// TwinCAT 3 PLC project Monolitico
// ProgramVersion: 3.1.4024.0
// libraries:
//   CmpBitmapPool, * (System)
//   Tc2_Standard, * (Beckhoff Automation GmbH)
//   Tc2_System, * (Beckhoff Automation GmbH)
//   Tc3_Module, * (Beckhoff Automation GmbH)
//   VisuDialogs, * (System)
// project tree:
//   / GlobalTextList.TcGTLO, PlcTask.TcTTO, Visualization Manager.TcVMO (not stored)
//   POUs/ FB_Bloque.TcPOU, MAIN.TcPOU
//   VISUs/ ImagePool.TcIPO (not stored), Visualization.TcVIS
// (motion and I/O tree: see PLC project manual)
// real-time tasks:
//   TASK PlcTask: cycle T#10ms, priority 20, ADS port 350
//   TASK PlcTask1: cycle T#10ms, priority 21, ADS port 351

CONFIGURATION Monolitico
    RESOURCE PLC ON TwinCAT3
        TASK PlcTask(INTERVAL := T#10ms, PRIORITY := 20);
        PROGRAM MAIN WITH PlcTask : MAIN;
    END_RESOURCE
END_CONFIGURATION

// ---- POUs/MAIN.TcPOU
PROGRAM MAIN
VAR
	
	//Pulsador AT %I*: BOOL;
	//Lampara AT %Q*: BOOL;
	
	Selector_modo_manual AT %I*: BOOL;
	
	test_pieza: FB_Bloque;

END_VAR

IF NOT Selector_modo_manual THEN
test_pieza();
END_IF

END_PROGRAM

// ---- POUs/FB_Bloque.TcPOU
FUNCTION_BLOCK FB_Bloque
VAR_INPUT
	Tcheck: TIME := T#1S;
	Treset: TIME := T#1S;
	Tdesplazador: TIME := T#1S;
	Tcinta: TIME := T#0.5S;
END_VAR
VAR_OUTPUT
END_VAR
VAR
	Ciclos: INT;
	Aceptados:INT;
	Rechazados: INT;
	Restantes: INT;
	
	pieza_ok: BOOL;
	
	//Terminal 2
	Pulsador_parada_emergencia AT %I*: BOOL;
	Selector_modo_manual AT %I*: BOOL;
	Pulsador_marcha AT %I*: BOOL;
	Pulsador_parada_NC AT %I*: BOOL;
	Parte_operativa_conectada AT %I*: BOOL;
	Presencia_pale AT %I*: BOOL;
	Codigo_pale_bit_0 AT %I*: BOOL;
	Codigo_pale_bit_1 AT %I*: BOOL;
	
	
	//Terminal 3
	Codigo_pale_bit_2 AT %I*: BOOL;
	Detector_presion AT %I*: BOOL;
	
	//Terminal 4
	Desconecta_parte_operativa AT %Q*: BOOL;
	Lampara_alarma AT %Q*: BOOL;
	Lampara_marcha AT %Q*: BOOL;
	Lampara_falta_material AT %Q*: BOOL;
	Activa_marcha_motor_cinta AT %Q*: BOOL;
	Invierte_marcha_motor_cinta AT %Q*: BOOL;
	Retenedor_pale_baja AT %Q*: BOOL;
	Separador_pale_sube AT %Q*: BOOL;
	
	
	//Terminal 5
 	Avisador_sonoro AT %Q*: BOOL;
	
	//Terminal 6
	Horizontal_descargador_detras AT %I*: BOOL;
	Horizontal_descargador_delante AT %I*: BOOL;
	Vertical_descargador_arriba AT %I*: BOOL;
	Vertical_descargador_abajo AT %I*: BOOL;
	Verificador_arriba AT %I*: BOOL;
	Verificador_abajo AT %I*: BOOL;
	Desplazador_detras AT %I*: BOOL;
	Alimentador_detras AT %I*: BOOL;
	
	
	//Terminal 7
	Alimentador_delante AT %I*: BOOL;
	Vacio_obtenido_vacuostato_descargador AT %I*: BOOL;
	Base_en_Alimentador AT %I*: BOOL;
	
	//Terminal 8
	Descargador_adelante AT %Q*: BOOL;
	Descargador_atras AT %Q*: BOOL;
	Descargador_baja AT %Q*: BOOL;
	Rechazador_adelante AT %Q*: BOOL;
	Verificador_baja AT %Q*: BOOL;
	Desplazador_adelante AT %Q*: BOOL;
	Alimentador_adelante AT %Q*: BOOL;
	Eyector_succiona AT %Q*: BOOL;
	
	NOLAMP: INT;
	t: INT;
	NOTSOUND: INT;
	NOTFOUND: INT;
END_VAR

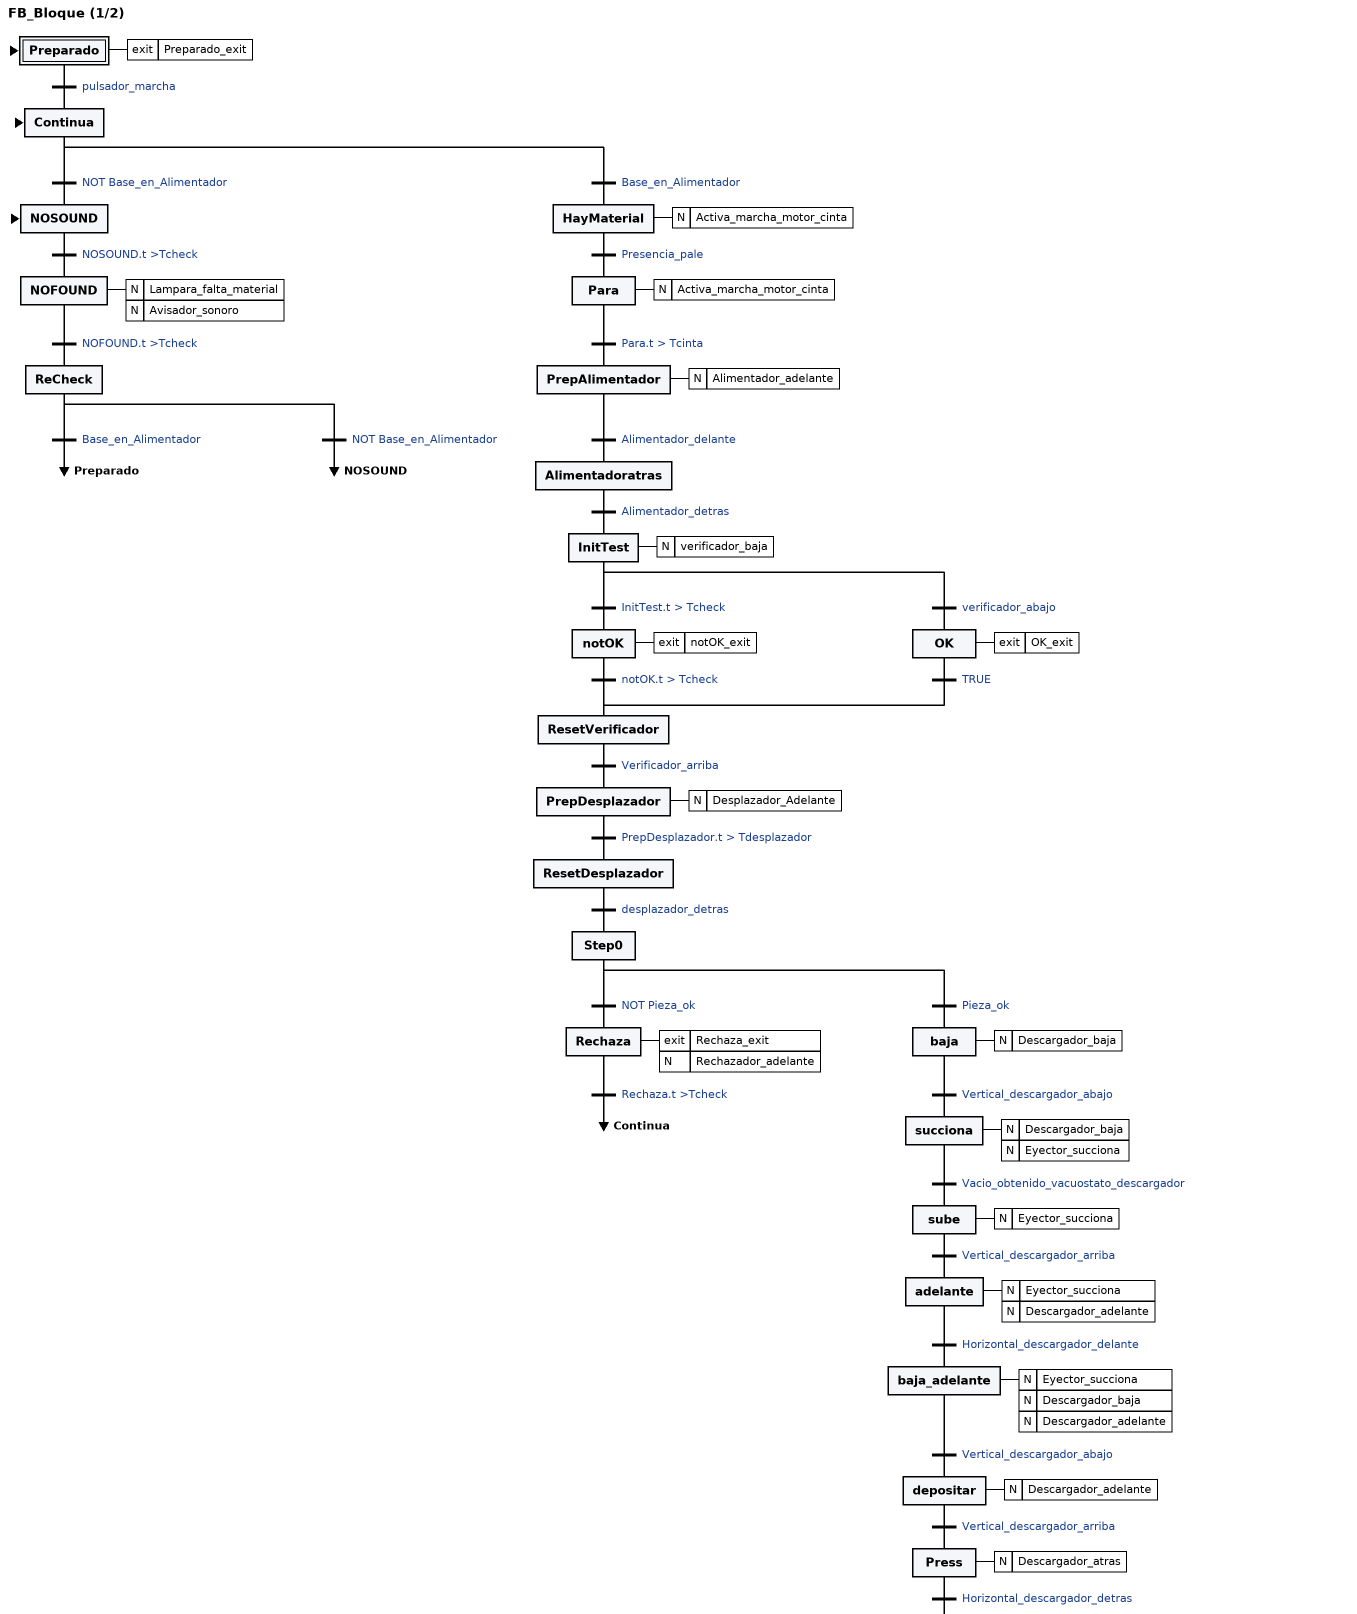
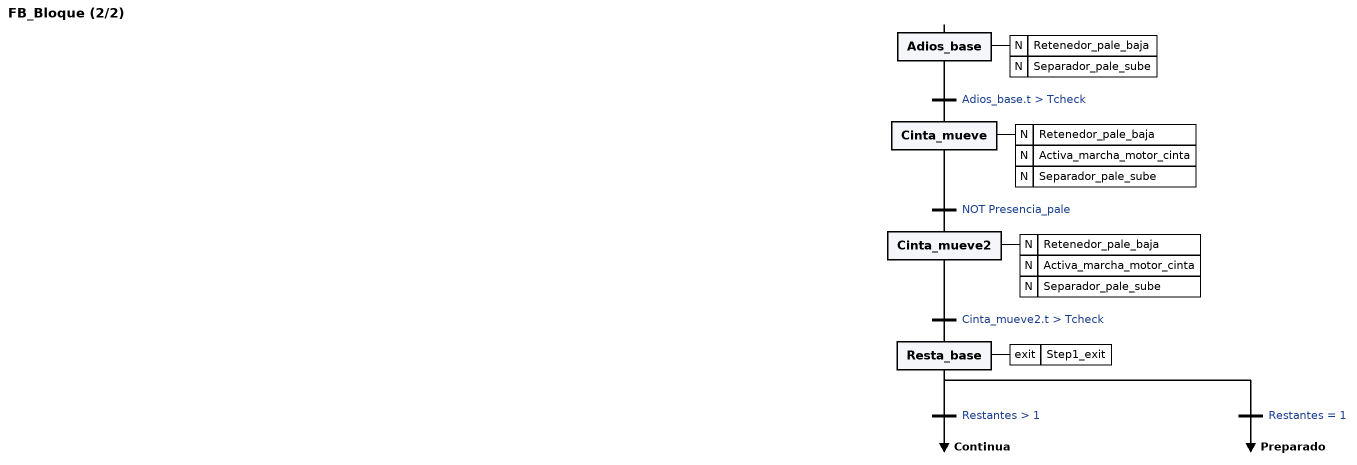
INITIAL_STEP Preparado:
    Preparado_exit(P0);  // exit action
END_STEP
TRANSITION FROM Preparado TO Continua
    := pulsador_marcha;
END_TRANSITION
STEP Continua:
END_STEP
TRANSITION FROM Continua TO NOSOUND
    := NOT Base_en_Alimentador;
END_TRANSITION
STEP NOSOUND:
END_STEP
TRANSITION FROM NOSOUND TO NOFOUND
    := NOSOUND.t >Tcheck;
END_TRANSITION
STEP NOFOUND:
    Lampara_falta_material(N);
    Avisador_sonoro(N);
END_STEP
TRANSITION FROM NOFOUND TO ReCheck
    := NOFOUND.t >Tcheck;
END_TRANSITION
STEP ReCheck:
END_STEP
TRANSITION FROM ReCheck TO Preparado
    := Base_en_Alimentador;
END_TRANSITION
TRANSITION FROM ReCheck TO NOSOUND
    := NOT Base_en_Alimentador;
END_TRANSITION
TRANSITION FROM Continua TO HayMaterial
    := Base_en_Alimentador;
END_TRANSITION
STEP HayMaterial:
    Activa_marcha_motor_cinta(N);
END_STEP
TRANSITION FROM HayMaterial TO Para
    := Presencia_pale;
END_TRANSITION
STEP Para:
    Activa_marcha_motor_cinta(N);
END_STEP
TRANSITION FROM Para TO PrepAlimentador
    := Para.t > Tcinta;
END_TRANSITION
STEP PrepAlimentador:
    Alimentador_adelante(N);
END_STEP
TRANSITION FROM PrepAlimentador TO Alimentadoratras
    := Alimentador_delante;
END_TRANSITION
STEP Alimentadoratras:
END_STEP
TRANSITION FROM Alimentadoratras TO InitTest
    := Alimentador_detras;
END_TRANSITION
STEP InitTest:
    verificador_baja(N);
END_STEP
TRANSITION FROM InitTest TO notOK
    := InitTest.t > Tcheck;
END_TRANSITION
STEP notOK:
    notOK_exit(P0);  // exit action
END_STEP
TRANSITION FROM notOK TO ResetVerificador
    := notOK.t > Tcheck;
END_TRANSITION
TRANSITION FROM InitTest TO OK
    := verificador_abajo;
END_TRANSITION
STEP OK:
    OK_exit(P0);  // exit action
END_STEP
TRANSITION FROM OK TO ResetVerificador
    := TRUE;
END_TRANSITION
STEP ResetVerificador:
END_STEP
TRANSITION FROM ResetVerificador TO PrepDesplazador
    := Verificador_arriba;
END_TRANSITION
STEP PrepDesplazador:
    Desplazador_Adelante(N);
END_STEP
TRANSITION FROM PrepDesplazador TO ResetDesplazador
    := PrepDesplazador.t > Tdesplazador;
END_TRANSITION
STEP ResetDesplazador:
END_STEP
TRANSITION FROM ResetDesplazador TO Step0
    := desplazador_detras;
END_TRANSITION
STEP Step0:
END_STEP
TRANSITION FROM Step0 TO Rechaza
    := NOT Pieza_ok;
END_TRANSITION
STEP Rechaza:
    Rechaza_exit(P0);  // exit action
    Rechazador_adelante(N);
END_STEP
TRANSITION FROM Rechaza TO Continua
    := Rechaza.t >Tcheck;
END_TRANSITION
TRANSITION FROM Step0 TO baja
    := Pieza_ok;
END_TRANSITION
STEP baja:
    Descargador_baja(N);
END_STEP
TRANSITION FROM baja TO succiona
    := Vertical_descargador_abajo;
END_TRANSITION
STEP succiona:
    Descargador_baja(N);
    Eyector_succiona(N);
END_STEP
TRANSITION FROM succiona TO sube
    := Vacio_obtenido_vacuostato_descargador;
END_TRANSITION
STEP sube:
    Eyector_succiona(N);
END_STEP
TRANSITION FROM sube TO adelante
    := Vertical_descargador_arriba;
END_TRANSITION
STEP adelante:
    Eyector_succiona(N);
    Descargador_adelante(N);
END_STEP
TRANSITION FROM adelante TO baja_adelante
    := Horizontal_descargador_delante;
END_TRANSITION
STEP baja_adelante:
    Eyector_succiona(N);
    Descargador_baja(N);
    Descargador_adelante(N);
END_STEP
TRANSITION FROM baja_adelante TO depositar
    := Vertical_descargador_abajo;
END_TRANSITION
STEP depositar:
    Descargador_adelante(N);
END_STEP
TRANSITION FROM depositar TO Press
    := Vertical_descargador_arriba;
END_TRANSITION
STEP Press:
    Descargador_atras(N);
END_STEP
TRANSITION FROM Press TO Adios_base
    := Horizontal_descargador_detras;
END_TRANSITION
STEP Adios_base:
    Retenedor_pale_baja(N);
    Separador_pale_sube(N);
END_STEP
TRANSITION FROM Adios_base TO Cinta_mueve
    := Adios_base.t > Tcheck;
END_TRANSITION
STEP Cinta_mueve:
    Retenedor_pale_baja(N);
    Activa_marcha_motor_cinta(N);
    Separador_pale_sube(N);
END_STEP
TRANSITION FROM Cinta_mueve TO Cinta_mueve2
    := NOT Presencia_pale;
END_TRANSITION
STEP Cinta_mueve2:
    Retenedor_pale_baja(N);
    Activa_marcha_motor_cinta(N);
    Separador_pale_sube(N);
END_STEP
TRANSITION FROM Cinta_mueve2 TO Resta_base
    := Cinta_mueve2.t > Tcheck;
END_TRANSITION
STEP Resta_base:
    Step1_exit(P0);  // exit action
END_STEP
TRANSITION FROM Resta_base TO Continua
    := Restantes > 1;
END_TRANSITION
TRANSITION FROM Resta_base TO Preparado
    := Restantes = 1;
END_TRANSITION

ACTION notOK_exit:
pieza_ok := FALSE;
END_ACTION

ACTION OK_exit:
pieza_ok := true;
END_ACTION

ACTION Preparado_entry:
//Ciclos:= 3;
Rechazados :=0;
Aceptados :=0;
Restantes:=Ciclos;
END_ACTION

ACTION Preparado_exit:
IF Restantes = 0 THEN

	Restantes := Ciclos;
	Aceptados := 0;
	Rechazados := 0;	

END_IF
END_ACTION

ACTION Rechaza_exit:
Rechazados:= Rechazados+1;
END_ACTION

ACTION Step1_exit:
Aceptados:=Aceptados+1;
Restantes:=Restantes-1;
END_ACTION

END_FUNCTION_BLOCK

// ---- GlobalTextList.TcGTLO
TEXTLIST GlobalTextList
  189 = '  ➡ ⬅ ⬇ ⬆ ← → ↓ ↑'
  198 = ' ➙'
  307 = '%i'
  729 = '0'
  472 = '1'
  731 = '<'
  44 = '>'
  12 = 'A+'
  482 = 'A-'
  789 = 'Abajo'
  231 = 'Aceptados'
  66 = 'Alarma'
  224 = 'Alimentador'
  25 = 'Arriba'
  54 = 'Aspirar'
  267 = 'B+'
  782 = 'B-'
  801 = 'C+'
  215 = 'C-'
  701 = 'Ciclos'
  642 = 'Ciclos Completados'
  957 = 'Cinta'
  81 = 'Colocado'
  497 = 'Comenzar'
  143 = 'D+'
  630 = 'D-'
  481 = 'Delante'
  437 = 'Descargador'
  936 = 'Desplazador'
  445 = 'Detrás'
  74 = 'E+'
  781 = 'E-'
  742 = 'E-Stop'
  908 = 'Estado'
  286 = 'Estoy Abajo'
  148 = 'Estoy Arriba'
  955 = 'Eyector'
  417 = 'F+'
  707 = 'F-'
  878 = 'FALTA M.'
  395 = 'FM'
  769 = 'FMS-201                                 ALIMENTADORA DE BASES                                                    VTL     '
  561 = 'Horizontal'
  750 = 'Lámpara'
  45 = 'Marcha'
  634 = 'Material'
  861 = 'Panel'
  463 = 'Parada'
  619 = 'pb'
  935 = 'Pieza NO OK'
  336 = 'Pieza OK'
  741 = 'Pieza Ok'
  524 = 'Planta'
  640 = 'pp'
  783 = 'Preparado'
  330 = 'R+'
  876 = 'Rechazador'
  970 = 'Rechazados'
  888 = 'Rechazads'
  94 = 'Rehczados'
  560 = 'Restantes'
  531 = 'Rev'
  452 = 'Run'
  784 = 'S+'
  815 = 'Succionar'
  643 = 'Tarea'
  710 = 'V+'
  288 = 'V-'
  629 = 'Vacío'
  125 = 'Verificador'
  839 = 'Verificador Activado'
  483 = 'Vertical'
  575 = '➡'
  509 = '⬅'
  381 = '⬆'
  169 = '⬇'
END_TEXTLIST

// ---- VISUs/Visualization.TcVIS
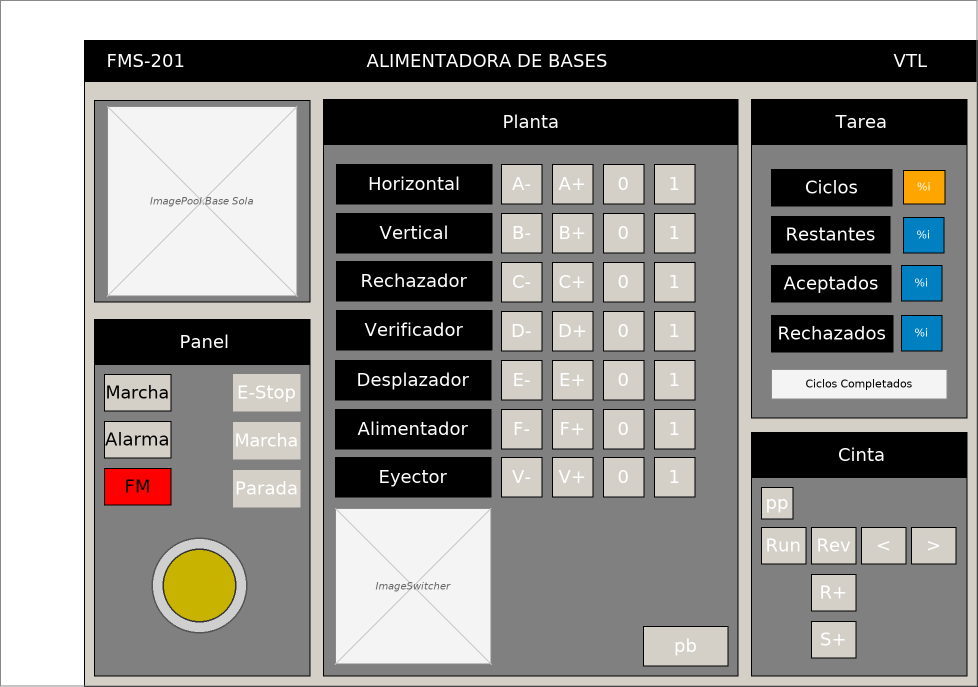
VISUALIZATION Visualization  // 978x687
    Rectangle (84,81 894x606)
    Rectangle (751,144 216x274)
    Rectangle (323,144 415x532)
    Rectangle (323,99 415x45)
    Label (323,101 416x42), "Planta"
    Rectangle (751,99 216x45)
    Label (801,104 121x36), "Tarea"
    Progressbar (771,369 176x30), "Ciclos Completados", variable: MAIN.test_pieza.Aceptados
    RoundedRectangle (336,164 156x40), "Horizontal", colour toggle: MAIN.test_pieza.Descargador_adelante
    Textfield (903,170 42x34), "%i", text variable: MAIN.test_pieza.Ciclos
        OnMouseDown: write MAIN.test_pieza.Ciclos via VisuDialogs.Numpad, min 1, max 10
    RoundedRectangle (771,169 121x37), "Ciclos"
    RoundedRectangle (771,216 119x37), "Restantes"
    RoundedRectangle (771,265 120x37), "Aceptados"
    RoundedRectangle (771,315 122x37), "Rechazados"
    Textfield (903,217 41x36), "%i", text variable: MAIN.test_pieza.Restantes
    Textfield (901,265 41x36), "%i", text variable: MAIN.test_pieza.Aceptados
    Textfield (901,315 41x36), "%i", text variable: MAIN.test_pieza.Rechazados
    RoundedRectangle (552,213 41x40), "B+", colour toggle: MAIN.test_pieza.Descargador_baja
        toggle MAIN.test_pieza.Descargador_baja
    Rectangle (751,477 216x199)
    Rectangle (751,432 216x45)
    Label (801,437 121x36), "Cinta"
    Rectangle (94,100 216x202)
    Rectangle (94,364 216x312)
    Rectangle (94,319 216x45)
    Label (144,324 121x36), "Panel"
    Rectangle (84,40 894x41)
    Label (84,41 893x40), "FMS-201 ALIMENTADORA DE BASES VTL"
    RoundedRectangle (336,213 156x40), "Vertical", colour toggle: MAIN.test_pieza.Descargador_adelante
    RoundedRectangle (552,164 41x40), "A+", colour toggle: MAIN.test_pieza.Descargador_adelante
        tap MAIN.test_pieza.Descargador_adelante
    RoundedRectangle (552,262 41x40), "C+", colour toggle: MAIN.test_pieza.Rechazador_adelante
        tap MAIN.test_pieza.Rechazador_adelante
    RoundedRectangle (552,311 41x40), "D+", colour toggle: MAIN.test_pieza.Verificador_baja
        tap MAIN.test_pieza.Verificador_baja
    RoundedRectangle (552,360 41x40), "E+", colour toggle: MAIN.test_pieza.Desplazador_adelante
        tap MAIN.test_pieza.Desplazador_adelante
    RoundedRectangle (552,409 41x40), "F+", colour toggle: MAIN.test_pieza.Alimentador_adelante
        tap MAIN.test_pieza.Alimentador_adelante
        toggle MAIN.test_pieza.Descargador_baja
    RoundedRectangle (552,457 41x40), "V+", colour toggle: MAIN.test_pieza.Eyector_succiona
        toggle MAIN.test_pieza.Eyector_succiona
    RoundedRectangle (336,261 156x40), "Rechazador", colour toggle: MAIN.test_pieza.Descargador_adelante
    RoundedRectangle (336,310 156x40), "Verificador", colour toggle: MAIN.test_pieza.Descargador_adelante
    RoundedRectangle (335,360 156x40), "Desplazador", colour toggle: MAIN.test_pieza.Descargador_adelante
    RoundedRectangle (335,409 156x40), "Alimentador", colour toggle: MAIN.test_pieza.Descargador_adelante
    RoundedRectangle (335,457 156x40), "Eyector", colour toggle: MAIN.test_pieza.Descargador_adelante
    RoundedRectangle (501,164 41x40), "A-", colour toggle: MAIN.test_pieza.Descargador_atras
        tap MAIN.test_pieza.Descargador_atras
    RoundedRectangle (603,164 41x40), "0", colour toggle: MAIN.test_pieza.Horizontal_descargador_detras
        tap MAIN.test_pieza.Horizontal_descargador_detras
    RoundedRectangle (654,164 41x40), "1", colour toggle: MAIN.test_pieza.Horizontal_descargador_delante
        tap MAIN.test_pieza.Horizontal_descargador_delante
    RoundedRectangle (603,213 41x40), "0", colour toggle: MAIN.test_pieza.Vertical_descargador_arriba
        tap MAIN.test_pieza.Vertical_descargador_arriba
    RoundedRectangle (654,213 41x40), "1", colour toggle: MAIN.test_pieza.Vertical_descargador_abajo
        tap MAIN.test_pieza.Vertical_descargador_abajo
    RoundedRectangle (603,262 41x40), "0"
    RoundedRectangle (603,311 41x40), "0", colour toggle: MAIN.test_pieza.Verificador_arriba
        tap MAIN.test_pieza.Verificador_arriba
    RoundedRectangle (603,360 41x40), "0", colour toggle: MAIN.test_pieza.Desplazador_detras
        tap MAIN.test_pieza.Desplazador_detras
    RoundedRectangle (603,409 41x40), "0", colour toggle: MAIN.test_pieza.Alimentador_detras
        tap MAIN.test_pieza.Alimentador_detras
    RoundedRectangle (603,457 41x40), "0"
    RoundedRectangle (654,262 41x40), "1"
    RoundedRectangle (654,311 41x40), "1", colour toggle: MAIN.test_pieza.Verificador_abajo
        tap MAIN.test_pieza.Verificador_abajo
    RoundedRectangle (654,360 41x40), "1"
    RoundedRectangle (654,409 41x40), "1", colour toggle: MAIN.test_pieza.Alimentador_delante
        tap MAIN.test_pieza.Alimentador_delante
    RoundedRectangle (654,457 41x40), "1", colour toggle: MAIN.test_pieza.Vacio_obtenido_vacuostato_descargador
        tap MAIN.test_pieza.Vacio_obtenido_vacuostato_descargador
    RoundedRectangle (501,213 41x40), "B-"
    RoundedRectangle (501,262 41x40), "C-"
    RoundedRectangle (501,311 41x40), "D-"
    RoundedRectangle (501,360 41x40), "E-"
    RoundedRectangle (501,409 41x40), "F-"
    RoundedRectangle (501,457 41x40), "V-"
    RoundedRectangle (643,626 85x40), "pb", colour toggle: MAIN.test_pieza.Base_en_Alimentador
        tap MAIN.test_pieza.Base_en_Alimentador
    RoundedRectangle (104,468 67x37), "FM", colour toggle: MAIN.test_pieza.Lampara_falta_material
        tap MAIN.test_pieza.Lampara_falta_material
    RoundedRectangle (761,487 32x32), "pp", colour toggle: MAIN.test_pieza.Presencia_pale
        tap MAIN.test_pieza.Presencia_pale
    RoundedRectangle (911,527 45x37), ">", colour toggle: MAIN.test_pieza.Activa_marcha_motor_cinta
        tap MAIN.test_pieza.Activa_marcha_motor_cinta
    RoundedRectangle (861,527 45x37), "<", colour toggle: MAIN.test_pieza.Invierte_marcha_motor_cinta
        toggle MAIN.test_pieza.Invierte_marcha_motor_cinta
    RoundedRectangle (761,527 45x37), "Run", colour toggle: MAIN.test_pieza.Activa_marcha_motor_cinta
    RoundedRectangle (811,527 45x37), "Rev", colour toggle: MAIN.test_pieza.Invierte_marcha_motor_cinta
    RoundedRectangle (811,574 45x37), "R+", colour toggle: MAIN.test_pieza.Retenedor_pale_baja
        tap MAIN.test_pieza.Retenedor_pale_baja
    RoundedRectangle (811,621 45x37), "S+", colour toggle: MAIN.test_pieza.Separador_pale_sube
        tap MAIN.test_pieza.Separador_pale_sube
    RoundedRectangle (233,374 67x37), "E-Stop", colour toggle: MAIN.test_pieza.Pulsador_parada_emergencia
        tap MAIN.test_pieza.Pulsador_parada_emergencia
    RoundedRectangle (233,422 67x37), "Marcha", colour toggle: MAIN.test_pieza.Pulsador_marcha
        tap MAIN.test_pieza.Pulsador_marcha
    RoundedRectangle (233,470 67x37), "Parada", colour toggle: MAIN.test_pieza.Pulsador_parada_NC
        tap MAIN.test_pieza.Pulsador_parada_NC
    RoundedRectangle (104,421 67x37), "Alarma", colour toggle: MAIN.test_pieza.Lampara_alarma
        tap MAIN.test_pieza.Lampara_alarma
    RoundedRectangle (104,374 67x37), "Marcha", colour toggle: MAIN.test_pieza.Lampara_marcha
        tap MAIN.test_pieza.Lampara_marcha
    Image (107,106 190x190), image: ImagePool.Base Sola
    Lamp1 (142,530 115x111), variable: MAIN.test_pieza.Lampara_falta_material, style: Lamp-Lamp1-Yellow
    ImageSwitcher (335,508 156x156), variable: MAIN.test_pieza.pieza_ok, background image: ImagePool.Base OK, image: ImagePool.Base No OK, behaviour: TOGGLE
END_VISUALIZATION
